// TwinCAT 3 PLC project Plc
// Title: Plc
// Company: Vortex.Library
// ProjectVersion: 1.9.6.256
// ProgramVersion: 3.1.4023.0
// libraries:
//   Tc2_Standard, * (Beckhoff Automation GmbH)
//   Tc2_System, * (Beckhoff Automation GmbH)
//   Tc3_Module, * (Beckhoff Automation GmbH)
// project tree:
//   / PlcTask.TcTTO (not stored)
//   POUs/ MAIN.TcPOU, stProduction.TcDUT, stStations.TcDUT
//   POUs/Stations/ stStationCu1.TcDUT, stStationCu2.TcDUT, stStationCu3.TcDUT, stStationCu4.TcDUT
//   POUs/Test/ stNested.TcDUT, stTestEnum.TcDUT
// real-time tasks:
//   TASK PlcTask: cycle T#10ms, priority 20, ADS port 350
//   TASK PlcTask1: cycle T#10ms, priority 21, ADS port 351

// ---- POUs/Stations/stStationCu1.TcDUT
TYPE stStationCu1 :
STRUCT
	{attribute addProperty Name "Name"}
	Name : STRING := 'Station 1';
	{attribute addProperty Name "Is On"}	
    IsOn : BOOL := TRUE;
	{attribute addProperty Name "Station status"}
	Cu1Enum : stTestEnum;
	{attribute addProperty Name "Time"}
	TimeOfDay: TIME_OF_DAY;
	{attribute addProperty Name "Date"}
    TestDate : DATE;	
	{attribute addProperty Name "Nested Station 1"}
	{attribute wpf [Container(Layout.Wrap)]}
	NestedFirst : stNested := (Name:='Nested Station 1', NestedOn := TRUE); 
	{attribute addProperty Name "Nested Station 2"}
	{attribute wpf [Container(Layout.Wrap)]}
	NestedSecond : stNested := (Name:='Nested Station 2'); 
END_STRUCT
END_TYPE

// ---- POUs/Stations/stStationCu2.TcDUT
TYPE stStationCu2 :
STRUCT
	{attribute addProperty Name "Name"}
	Name : STRING := 'Station 2';
	{attribute addProperty Name "Is On"}	
    IsOn : BOOL := TRUE;
	{attribute addProperty Name "Station status"}
	Cu1Enum : stTestEnum := 1;
	{attribute addProperty Name "Time"}
	TimeOfDay: TIME_OF_DAY;
	{attribute addProperty Name "Date"}
    TestDate : DATE;	 
	{attribute addProperty Name "Nested Element"}
	{attribute wpf [Container(Layout.Wrap)]}
	Complex : stNested := (Name:='Nested Station 1',NestedOn := TRUE); 
END_STRUCT
END_TYPE

// ---- POUs/Stations/stStationCu3.TcDUT
TYPE stStationCu3 :
STRUCT
	{attribute addProperty Name "Name"}
	Name : STRING := 'Station 3';
	{attribute addProperty Name "Is On"}	
    IsOn : BOOL;
	{attribute addProperty Name "Station status"}
	Cu1Enum : stTestEnum;
	{attribute addProperty Name "Time"}
	TimeOfDay: TIME_OF_DAY;
	{attribute addProperty Name "Date"}
    TestDate : DATE;	 
END_STRUCT
END_TYPE

// ---- POUs/Stations/stStationCu4.TcDUT
TYPE stStationCu4 :
STRUCT
	{attribute addProperty Name "Name"}
	Name : STRING := 'Station 4';
	{attribute addProperty Name "Is On"}	
    IsOn : BOOL;
	{attribute addProperty Name "Station status"}
	Cu1Enum : stTestEnum;
	{attribute addProperty Name "Time"}
	TimeOfDay: TIME_OF_DAY;
	{attribute addProperty Name "Date"}
    TestDate : DATE;	 
END_STRUCT
END_TYPE

// ---- POUs/stProduction.TcDUT
TYPE stProduction :
STRUCT
	

	ok_pieces : INT := 0;
	
	nok_pieces : INT := 0;
	
	start : BOOL;
	
	{attribute addProperty Name "<#Integer From PLC#>"}	
	progress_bar_value : INT;
	{attribute addProperty Name "<#Bool From PLC#>"}	
    progress_bar_status : BOOL;
	
END_STRUCT
END_TYPE

// ---- POUs/stStations.TcDUT
{attribute wpf [Container(Layout.Tabs)]}
TYPE stStations :
STRUCT
	{attribute addProperty Name "Station1"}
	stationCu1 : stStationCu1;
	{attribute addProperty Name "Station2"}
	stationCu2 : stStationCu2;
	{attribute addProperty Name "Station3"}
	stationCu3 : stStationCu3;
	{attribute addProperty Name "Station4"}
	stationCu4 : stStationCu4;
END_STRUCT
END_TYPE

// ---- POUs/Test/stNested.TcDUT
TYPE stNested :
STRUCT
	{attribute addProperty Name "Name"}
	Name : STRING;
	{attribute addProperty Name "Turn on nested station"}
	NestedOn : BOOL;	
	{attribute addProperty Name "Date and Time"}
	TestDateTime : DATE_AND_TIME;	
END_STRUCT
END_TYPE

// ---- POUs/Test/stTestEnum.TcDUT
{attribute 'qualified_only'}
{attribute 'strict'}
TYPE stTestEnum :
(
	Unknown := 0,
	Available := 1,
	UnAvailable := 2	
);
END_TYPE

// ---- POUs/MAIN.TcPOU
PROGRAM MAIN
VAR
	
	
	{attribute addProperty Name "<#Hello#> <#World#>"}
	Hello_World : STRING;
	
    stations : stStations;
	
	production : stProduction;
	
	

	
END_VAR

Hello_World := 'This is automatically generated UI!' ;
IF production.progress_bar_status = TRUE THEN
	production.progress_bar_value := production.progress_bar_value + 1;
	
	IF production.progress_bar_value MOD 10 = 0 THEN
		production.ok_pieces := production.ok_pieces + 1 ;
	END_IF
	
	IF production.progress_bar_value MOD 100 = 0 THEN
		production.nok_pieces := production.nok_pieces + 1 ;
	END_IF
	IF production.progress_bar_value = 1000 THEN
		production.progress_bar_status := FALSE; 
		
	END_IF
END_IF

END_PROGRAM
